// TIA Portal V16 export
// export: Created 2024-06-24T15:42:28.7695061Z, ExportSetting WithDefaults, DisplayName Totally Integrated Automation Portal, DisplayVersion V16, DisplayName TIA Portal Version Control Interface, DisplayVersion V16, DisplayName TIA Portal Openness, DisplayVersion V16, DisplayName STEP 7 Professional, DisplayVersion V16, DisplayName STEP 7 Safety, DisplayVersion V16, DisplayName WinCC Advanced, DisplayVersion V16
VAR_GLOBAL   // PLC tag table "Standard-Variablentabelle"
   "Belt Conveyor (4m) 0 Encoder Signal A" AT %I0.0 : Bool;
   "Retroreflective Sensor 0" AT %I0.1 : Bool;
   "Retroreflective Sensor 1" AT %I0.2 : Bool;
   "Diffuse Sensor 0" AT %I0.3 : Bool;
   Clock_Byte AT %MB0 : Byte;
   Clock_10Hz AT %M0.0 : Bool;
   Clock_5Hz AT %M0.1 : Bool;
   "Clock_2.5Hz" AT %M0.2 : Bool;
   Clock_2Hz AT %M0.3 : Bool;
   "Clock_1.25Hz" AT %M0.4 : Bool;
   Clock_1Hz AT %M0.5 : Bool;
   "Clock_0.625Hz" AT %M0.6 : Bool;
   "Clock_0.5Hz" AT %M0.7 : Bool;
   "Diffuse Sensor 1" AT %I0.4 : Bool;
   "Diffuse Sensor 2" AT %I0.5 : Bool;
   "Diffuse Sensor 3" AT %I0.6 : Bool;
   "Belt Conveyor (2m) 0" AT %Q0.0 : Bool;
   "Belt Conveyor (2m) 1" AT %Q0.1 : Bool;
   "Belt Conveyor (2m) 2" AT %Q0.2 : Bool;
   "Belt Conveyor (2m) 3" AT %Q0.3 : Bool;
   "Belt Conveyor (4m) 0" AT %Q0.4 : Bool;
   "Conveyor Scale 0 (+)" AT %Q0.5 : Bool;
   "Pop Up Wheel Sorter 0 (+)" AT %Q0.6 : Bool;
   "Pop Up Wheel Sorter 0 (Left)" AT %Q0.7 : Bool;
   "Pop Up Wheel Sorter 0 (Right)" AT %Q1.0 : Bool;
   "Vision Sensor 0" AT %ID30 : DInt;
   Factory_Running AT %I0.7 : Bool;
   "Emergency Stop 0" AT %I1.0 : Bool;
   "Selector 0 (State 0)" AT %I1.1 : Bool;
   "Start Button 0" AT %I1.2 : Bool;
   "Two-Axis Pick & Place 0 (Detected)" AT %I1.3 : Bool;
   "Two-Axis Pick & Place 0 (Moving X)" AT %I1.4 : Bool;
   "Two-Axis Pick & Place 0 (Moving Z)" AT %I1.5 : Bool;
   "Two-Axis Pick & Place 0 X" AT %Q1.1 : Bool;
   "Two-Axis Pick & Place 0 Z" AT %Q1.2 : Bool;
   "Two-Axis Pick & Place 0 (Grab)" AT %Q1.3 : Bool;
   "Conveyor Scale 0 Weight (V)" AT %ID42 : Real;
   "Diffuse Sensor 4" AT %I1.6 : Bool;
   "Diffuse Sensor 6" AT %I1.7 : Bool;
   "Diffuse Sensor 5" AT %I2.0 : Bool;
   System_Byte AT %MB1 : Byte;
   FirstScan AT %M1.0 : Bool;
   DiagStatusUpdate AT %M1.1 : Bool;
   AlwaysTRUE AT %M1.2 : Bool;
   AlwaysFALSE AT %M1.3 : Bool;
END_VAR
